# EPICS substitutions: apps/mmfeuApp/Db/mmfeucrateAHDC.substitutions
file "db/mmfeucrate.db" {
        pattern { P, C, PORT}
                {"B_DET_AHDC_FEU", "1", "L1"  }
                {"B_DET_AHDC_FEU", "2", "L1"  }
                {"B_DET_AHDC_FEU", "3", "L1"  }
}
